(* IEC 61131-3 sources: POMIRTS_lab3/AS/Library_2/ArUnitConv, 3 files *)

(* ---- ArUnitConv.typ ---- *)
TYPE
	ArUnitConvAsyncInternalType : STRUCT
        FBStateCtx		: ArFBStateInternalType;
		AsyFuMaCtx		: ArFBAsyFuMaInternalType;
	END_STRUCT;
END_TYPE

(* ---- ArUnitConv.fun ---- *)
{REDUND_CONTEXT} {REDUND_UNREPLICABLE} FUNCTION_BLOCK ArUnitConvIsConvertible		(*Checks if units are convertible*)
	VAR_INPUT
		Execute					: BOOL;			(*Start execution.*)
		InputUnitID				: UDINT;		(*Identifier of input unit.*)
		InputUnitNamespaceID	: UDINT;		(*Identifier of input unit namespace, 0 for default namespace.*)
		OutputUnitID			: UDINT;		(*Identifier of output unit.*)
		OutputUnitNamespaceID	: UDINT;		(*Identifier of output unit namespace, 0 for default namespace.*)
	END_VAR
	VAR_OUTPUT
		Done					: BOOL;			(*Execution done.*)
		Busy					: BOOL;			(*Execution running.*)
		Error					: BOOL;			(*Execution failed.*)
		StatusID		 		: DINT;			(*Execution error: see help.*)
		Convertible				: BOOL;			(*Returns TRUE when the units are convertible, FALSE if not.*)
	END_VAR
	VAR
        Internal				: ArUnitConvAsyncInternalType;		(*Internal variable.*)
	END_VAR
END_FUNCTION_BLOCK

{REDUND_CONTEXT} {REDUND_UNREPLICABLE} FUNCTION_BLOCK ArUnitConvConvert		(*Converts a value from one unit to another.*)
	VAR_INPUT
		Execute					: BOOL;			(*Start execution.*)
		InputUnitID				: UDINT;		(*Identifier of input unit.*)
		InputUnitNamespaceID	: UDINT;		(*Identifier of input unit namespace, 0 for default namespace.*)
		OutputUnitID			: UDINT;		(*Identifier of output unit.*)
		OutputUnitNamespaceID	: UDINT;		(*Identifier of output unit namespace, 0 for default namespace.*)
		InputValue				: LREAL;		(*Value for conversion.*)
	END_VAR
	VAR_OUTPUT
		Done					: BOOL;			(*Execution done.*)
		Busy					: BOOL;         (*Execution running.*)
		Error					: BOOL;         (*Execution failed.*)
		StatusID		 		: DINT;			(*Execution error: see help.*)
		OutputValue				: LREAL;		(*Converted value.*)
	END_VAR
	VAR
        Internal				: ArUnitConvAsyncInternalType;		(*Internal variable.*)
	END_VAR
END_FUNCTION_BLOCK

{REDUND_CONTEXT} {REDUND_UNREPLICABLE} FUNCTION_BLOCK ArUnitConvCommonCodeToUnitID		(*Converts the common code of an unit to its identifier.*)
	VAR_INPUT
		Execute			: BOOL;				(*Start execution.*)
		CommonCode		: STRING[3];		(*Common code.*)
	END_VAR
	VAR_OUTPUT
		Done					: BOOL;		(*Execution done.*)
		Busy					: BOOL;     (*Execution running.*)
		Error					: BOOL;     (*Execution failed.*)
		StatusID		 		: DINT;	    (*Execution error: see help.*)
		UnitID					: UDINT;    (*Unit identifier.*)
	END_VAR
	VAR
        Internal				: ArUnitConvAsyncInternalType;		(*Internal variable.*)
	END_VAR
END_FUNCTION_BLOCK

{REDUND_CONTEXT} {REDUND_UNREPLICABLE} FUNCTION_BLOCK ArUnitConvGetNamespaceID		(*Converts the namespace string to a namespace identifier*)
	VAR_INPUT
		Execute			: BOOL;				(*Start execution.*)
		Namespace		: UDINT;			(*Pointer to a string containing the namespace.*)
	END_VAR
	VAR_OUTPUT
		Done					: BOOL;		(*Execution done.*)
		Busy					: BOOL;     (*Execution running.*)
		Error					: BOOL;     (*Execution failed.*)
		StatusID		 		: DINT;	    (*Execution error: see help.*)
		NamespaceID				: USINT;    (*Namespace identifier.*)
	END_VAR
	VAR
        Internal				: ArUnitConvAsyncInternalType;		(*Internal Variable.*)
	END_VAR
END_FUNCTION_BLOCK

(* ---- ArUnitConv.var ---- *)
VAR CONSTANT
	arUNITCONV_ERR_INVALID_UNITID		: DINT := -1070585696;		(*Invalid unit identifier.*)
	arUNITCONV_ERR_INVALID_CC			: DINT := -1070585695;      (*Invalid common code.*)
	arUNITCONV_ERR_INVALID_NS			: DINT := -1070585694;      (*Invalid unit namespace.*)
	arUNITCONV_ERR_INVALID_NSID			: DINT := -1070585693;      (*Invalid namespace identifier.*)
	arUNITCONV_ERR_NOT_CONVERTIBLE		: DINT := -1070585692;      (*The units are not convertible.*)
	arUNITCONV_ERR_WRONG_DB				: DINT := -1070585691;      (*Unit database is corrupt or has an unsupported format.*)
	arUNITCONV_ERR_NO_DB				: DINT := -1070585690;		(*An internal error has occurred. Please contact B+R support.*)
	arUNITCONV_ERR_INTERNAL				: DINT := -1070585689;		(*An internal error has occurred. Please contact B+R support.*)
END_VAR
